Universal Robots URScript: tcpMov.script

def tcpMov(vect):

    # FeaturePose is the pose for the feature
    # vect = p[0.1, 0, 0, 0, 0, 0] makes us move 10cm in the X direction of the feature
    # credits: https://forum.universal-robots.com/t/move-tcp-relative-to-feature/15492

   tcp_pose = get_actual_tcp_pose()
   return pose_add(tcp_pose, vect)


end
